Staubli VAL3: make_if.pgx

program make_if(string& x_sItem)
  local string l_sMessage
  local num i
  local num l_nValue
  local string l_sEmpty
  local string l_sItem
  local num l_nSizeList
  local string l_sEvent
  local bool l_bActive
  local string l_sItemList
  local num l_nKey
  local num l_nIndex
  local string l_sButton[2]
  local bool l_bYes
begin
  //
  cls()
  // Select the operator
  call language:message(l_sMessage,110)
  call use:questionDialog(l_sMessage,saveInOut:sCondition,i)
  //
  // != >= > < <= ==
  // compose the istruction
  if i>=1 and i<=size(saveInOut:sCondition)
    x_sItem=x_sItem+saveInOut:sCondition[i-1]
  else
    // escape
    x_sItem=""
    return
  endIf
  // modify the actual item
  call use:type(2,12,x_sItem)
  // insert a value
  call language:message(l_sMessage,112)
  // get the yes_no button Key
  call language:getYesNo(l_sButton)
  // ask the question
  call use:yes_no(l_sMessage,l_sButton,l_bYes)
  // check it
  if l_bYes
    //
    // reuse the operator
    //
    call saveInOut:getSize_num(l_nSizeList)
    call getType(l_sItem)
    call use:setSizeList(21,0,17,10)
    call use:listcreate(l_sItem)
    // insert in the list
    for i=0 to l_nSizeList-1
      call saveInOut:get_num(l_sItemList,i)
      call isActive(l_bActive,l_sItemList)
      if l_bActive
        call use:listadd(l_sItemList)
      endIf
    endFor
    call use:listredraw(0)
    do
      // get the key
      l_nKey=get()
      // get one input from the list
      call use:listevent(l_nKey,l_nIndex,l_sEvent)
      if l_nKey==255
        return
      endIf
    until l_nKey==270
    // check if an item has been selected
    if l_sEvent==""
      x_sItem=""
      return
    else
      x_sItem=x_sItem+"NUM "+ l_sEvent
    endIf
  else
    // use a value
    call use:changeValue(l_nValue,-10000,10000,2+len(x_sItem),12,l_sEmpty)
    x_sItem=x_sItem+toString("",l_nValue)
  endIf
  // validate
  if use:bUseEscape
    x_sItem=""
  endIf
end
